      moveJ p935,v100,fine,tool1\WObj:=wobj0;
      moveJ p936,v100,fine,tool1\WObj:=wobj0;
      moveJ p937,v100,fine,tool1\WObj:=wobj0;
      moveJ p938,v100,fine,tool1\WObj:=wobj0;
      moveJ p939,v100,fine,tool1\WObj:=wobj0;
      moveJ p940,v100,fine,tool1\WObj:=wobj0;
      moveJ p941,v100,fine,tool1\WObj:=wobj0;
      moveJ p942,v100,fine,tool1\WObj:=wobj0;
      moveJ p943,v100,fine,tool1\WObj:=wobj0;
      moveJ p944,v100,fine,tool1\WObj:=wobj0;
      moveJ p945,v100,fine,tool1\WObj:=wobj0;
      moveJ p946,v100,fine,tool1\WObj:=wobj0;
      moveJ p947,v100,fine,tool1\WObj:=wobj0;
      moveJ p948,v100,fine,tool1\WObj:=wobj0;
      moveJ p949,v100,fine,tool1\WObj:=wobj0;
      moveJ p950,v100,fine,tool1\WObj:=wobj0;
      moveJ p951,v100,fine,tool1\WObj:=wobj0;
      moveJ p952,v100,fine,tool1\WObj:=wobj0;
      moveJ p953,v100,fine,tool1\WObj:=wobj0;
      moveJ p954,v100,fine,tool1\WObj:=wobj0;
      moveJ p955,v100,fine,tool1\WObj:=wobj0;
      moveJ p956,v100,fine,tool1\WObj:=wobj0;
      moveJ p957,v100,fine,tool1\WObj:=wobj0;
      moveJ p958,v100,fine,tool1\WObj:=wobj0;
      moveJ p959,v100,fine,tool1\WObj:=wobj0;
      moveJ p960,v100,fine,tool1\WObj:=wobj0;
      moveJ p961,v100,fine,tool1\WObj:=wobj0;
      moveJ p962,v100,fine,tool1\WObj:=wobj0;
      moveJ p963,v100,fine,tool1\WObj:=wobj0;
      moveJ p964,v100,fine,tool1\WObj:=wobj0;
      moveJ p965,v100,fine,tool1\WObj:=wobj0;
      moveJ p966,v100,fine,tool1\WObj:=wobj0;
      moveJ p967,v100,fine,tool1\WObj:=wobj0;
      moveJ p968,v100,fine,tool1\WObj:=wobj0;
      moveJ p969,v100,fine,tool1\WObj:=wobj0;
      moveJ p970,v100,fine,tool1\WObj:=wobj0;
      moveJ p971,v100,fine,tool1\WObj:=wobj0;
      moveJ p972,v100,fine,tool1\WObj:=wobj0;
      moveJ p973,v100,fine,tool1\WObj:=wobj0;
      moveJ p974,v100,fine,tool1\WObj:=wobj0;
      moveJ p975,v100,fine,tool1\WObj:=wobj0;
      moveJ p976,v100,fine,tool1\WObj:=wobj0;
      moveJ p977,v100,fine,tool1\WObj:=wobj0;
      moveJ p978,v100,fine,tool1\WObj:=wobj0;
      moveJ p979,v100,fine,tool1\WObj:=wobj0;
      moveJ p980,v100,fine,tool1\WObj:=wobj0;
      moveJ p981,v100,fine,tool1\WObj:=wobj0;
      moveJ p982,v100,fine,tool1\WObj:=wobj0;
      moveJ p983,v100,fine,tool1\WObj:=wobj0;
      moveJ p984,v100,fine,tool1\WObj:=wobj0;
      moveJ p985,v100,fine,tool1\WObj:=wobj0;
      moveJ p986,v100,fine,tool1\WObj:=wobj0;
      moveJ p987,v100,fine,tool1\WObj:=wobj0;
      moveJ p988,v100,fine,tool1\WObj:=wobj0;
      moveJ p989,v100,fine,tool1\WObj:=wobj0;
      moveJ p990,v100,fine,tool1\WObj:=wobj0;
      moveJ p991,v100,fine,tool1\WObj:=wobj0;
      moveJ p992,v100,fine,tool1\WObj:=wobj0;
      moveJ p993,v100,fine,tool1\WObj:=wobj0;
      moveJ p994,v100,fine,tool1\WObj:=wobj0;
      moveJ p995,v100,fine,tool1\WObj:=wobj0;
      moveJ p996,v100,fine,tool1\WObj:=wobj0;
      moveJ p997,v100,fine,tool1\WObj:=wobj0;
      moveJ p998,v100,fine,tool1\WObj:=wobj0;
      moveJ p999,v100,fine,tool1\WObj:=wobj0;
      moveJ p1000,v100,fine,tool1\WObj:=wobj0;
      moveJ p1001,v100,fine,tool1\WObj:=wobj0;
      moveJ p1002,v100,fine,tool1\WObj:=wobj0;
      moveJ p1003,v100,fine,tool1\WObj:=wobj0;
      moveJ p1004,v100,fine,tool1\WObj:=wobj0;
      moveJ p1005,v100,fine,tool1\WObj:=wobj0;
      moveJ p1006,v100,fine,tool1\WObj:=wobj0;
      moveJ p1007,v100,fine,tool1\WObj:=wobj0;
      moveJ p1008,v100,fine,tool1\WObj:=wobj0;
      moveJ p1009,v100,fine,tool1\WObj:=wobj0;
      moveJ p1010,v100,fine,tool1\WObj:=wobj0;
      moveJ p1011,v100,fine,tool1\WObj:=wobj0;
      moveJ p1012,v100,fine,tool1\WObj:=wobj0;
      moveJ p1013,v100,fine,tool1\WObj:=wobj0;
      moveJ p1014,v100,fine,tool1\WObj:=wobj0;
      moveJ p1015,v100,fine,tool1\WObj:=wobj0;
      moveJ p1016,v100,fine,tool1\WObj:=wobj0;
      moveJ p1017,v100,fine,tool1\WObj:=wobj0;
      moveJ p1018,v100,fine,tool1\WObj:=wobj0;
      moveJ p1019,v100,fine,tool1\WObj:=wobj0;
      moveJ p1020,v100,fine,tool1\WObj:=wobj0;
      moveJ p1021,v100,fine,tool1\WObj:=wobj0;
      moveJ p1022,v100,fine,tool1\WObj:=wobj0;
      moveJ p1023,v100,fine,tool1\WObj:=wobj0;
      moveJ p1024,v100,fine,tool1\WObj:=wobj0;
      moveJ p1025,v100,fine,tool1\WObj:=wobj0;
      moveJ p1026,v100,fine,tool1\WObj:=wobj0;
      moveJ p1027,v100,fine,tool1\WObj:=wobj0;
      moveJ p1028,v100,fine,tool1\WObj:=wobj0;
      moveJ p1029,v100,fine,tool1\WObj:=wobj0;
      moveJ p1030,v100,fine,tool1\WObj:=wobj0;
      moveJ p1031,v100,fine,tool1\WObj:=wobj0;
      moveJ p1032,v100,fine,tool1\WObj:=wobj0;
      moveJ p1033,v100,fine,tool1\WObj:=wobj0;
      moveJ p1034,v100,fine,tool1\WObj:=wobj0;
      moveJ p1035,v100,fine,tool1\WObj:=wobj0;
      moveJ p1036,v100,fine,tool1\WObj:=wobj0;
      moveJ p1037,v100,fine,tool1\WObj:=wobj0;
      moveJ p1038,v100,fine,tool1\WObj:=wobj0;
      moveJ p1039,v100,fine,tool1\WObj:=wobj0;
      moveJ p1040,v100,fine,tool1\WObj:=wobj0;
      moveJ p1041,v100,fine,tool1\WObj:=wobj0;
      moveJ p1042,v100,fine,tool1\WObj:=wobj0;
      moveJ p1043,v100,fine,tool1\WObj:=wobj0;
      moveJ p1044,v100,fine,tool1\WObj:=wobj0;
      moveJ p1045,v100,fine,tool1\WObj:=wobj0;
      moveJ p1046,v100,fine,tool1\WObj:=wobj0;
      moveJ p1047,v100,fine,tool1\WObj:=wobj0;
      moveJ p1048,v100,fine,tool1\WObj:=wobj0;
      moveJ p1049,v100,fine,tool1\WObj:=wobj0;
      moveJ p1050,v100,fine,tool1\WObj:=wobj0;
      moveJ p1051,v100,fine,tool1\WObj:=wobj0;
      moveJ p1052,v100,fine,tool1\WObj:=wobj0;
      moveJ p1053,v100,fine,tool1\WObj:=wobj0;
      moveJ p1054,v100,fine,tool1\WObj:=wobj0;
      moveJ p1055,v100,fine,tool1\WObj:=wobj0;
      moveJ p1056,v100,fine,tool1\WObj:=wobj0;
      moveJ p1057,v100,fine,tool1\WObj:=wobj0;
      moveJ p1058,v100,fine,tool1\WObj:=wobj0;
      moveJ p1059,v100,fine,tool1\WObj:=wobj0;
      moveJ p1060,v100,fine,tool1\WObj:=wobj0;
      moveJ p1061,v100,fine,tool1\WObj:=wobj0;
      moveJ p1062,v100,fine,tool1\WObj:=wobj0;
      moveJ p1063,v100,fine,tool1\WObj:=wobj0;
      moveJ p1064,v100,fine,tool1\WObj:=wobj0;
      moveJ p1065,v100,fine,tool1\WObj:=wobj0;
      moveJ p1066,v100,fine,tool1\WObj:=wobj0;
      moveJ p1067,v100,fine,tool1\WObj:=wobj0;
      moveJ p1068,v100,fine,tool1\WObj:=wobj0;
      moveJ p1069,v100,fine,tool1\WObj:=wobj0;
      moveJ p1070,v100,fine,tool1\WObj:=wobj0;
      moveJ p1071,v100,fine,tool1\WObj:=wobj0;
      moveJ p1072,v100,fine,tool1\WObj:=wobj0;
      moveJ p1073,v100,fine,tool1\WObj:=wobj0;
      moveJ p1074,v100,fine,tool1\WObj:=wobj0;
      moveJ p1075,v100,fine,tool1\WObj:=wobj0;
      moveJ p1076,v100,fine,tool1\WObj:=wobj0;
      moveJ p1077,v100,fine,tool1\WObj:=wobj0;
      moveJ p1078,v100,fine,tool1\WObj:=wobj0;
      moveJ p1079,v100,fine,tool1\WObj:=wobj0;
      moveJ p1080,v100,fine,tool1\WObj:=wobj0;
      moveJ p1081,v100,fine,tool1\WObj:=wobj0;
      moveJ p1082,v100,fine,tool1\WObj:=wobj0;
      moveJ p1083,v100,fine,tool1\WObj:=wobj0;
      moveJ p1084,v100,fine,tool1\WObj:=wobj0;
      moveJ p1085,v100,fine,tool1\WObj:=wobj0;
      moveJ p1086,v100,fine,tool1\WObj:=wobj0;
      moveJ p1087,v100,fine,tool1\WObj:=wobj0;
      moveJ p1088,v100,fine,tool1\WObj:=wobj0;
      moveJ p1089,v100,fine,tool1\WObj:=wobj0;
      moveJ p1090,v100,fine,tool1\WObj:=wobj0;
      moveJ p1091,v100,fine,tool1\WObj:=wobj0;
      moveJ p1092,v100,fine,tool1\WObj:=wobj0;
      moveJ p1093,v100,fine,tool1\WObj:=wobj0;
      moveJ p1094,v100,fine,tool1\WObj:=wobj0;
      moveJ p1095,v100,fine,tool1\WObj:=wobj0;
      moveJ p1096,v100,fine,tool1\WObj:=wobj0;
      moveJ p1097,v100,fine,tool1\WObj:=wobj0;
      moveJ p1098,v100,fine,tool1\WObj:=wobj0;
      moveJ p1099,v100,fine,tool1\WObj:=wobj0;
      moveJ p1100,v100,fine,tool1\WObj:=wobj0;
      moveJ p1101,v100,fine,tool1\WObj:=wobj0;
      moveJ p1102,v100,fine,tool1\WObj:=wobj0;
      moveJ p1103,v100,fine,tool1\WObj:=wobj0;
      moveJ p1104,v100,fine,tool1\WObj:=wobj0;
      moveJ p1105,v100,fine,tool1\WObj:=wobj0;
      moveJ p1106,v100,fine,tool1\WObj:=wobj0;
      moveJ p1107,v100,fine,tool1\WObj:=wobj0;
      moveJ p1108,v100,fine,tool1\WObj:=wobj0;
      moveJ p1109,v100,fine,tool1\WObj:=wobj0;
      moveJ p1110,v100,fine,tool1\WObj:=wobj0;
      moveJ p1111,v100,fine,tool1\WObj:=wobj0;
      moveJ p1112,v100,fine,tool1\WObj:=wobj0;
      moveJ p1113,v100,fine,tool1\WObj:=wobj0;
      moveJ p1114,v100,fine,tool1\WObj:=wobj0;
      moveJ p1115,v100,fine,tool1\WObj:=wobj0;
      moveJ p1116,v100,fine,tool1\WObj:=wobj0;
      moveJ p1117,v100,fine,tool1\WObj:=wobj0;
      moveJ p1118,v100,fine,tool1\WObj:=wobj0;
      moveJ p1119,v100,fine,tool1\WObj:=wobj0;
      moveJ p1120,v100,fine,tool1\WObj:=wobj0;
      moveJ p1121,v100,fine,tool1\WObj:=wobj0;
      moveJ p1122,v100,fine,tool1\WObj:=wobj0;
      moveJ p1123,v100,fine,tool1\WObj:=wobj0;
      moveJ p1124,v100,fine,tool1\WObj:=wobj0;
      moveJ p1125,v100,fine,tool1\WObj:=wobj0;
      moveJ p1126,v100,fine,tool1\WObj:=wobj0;
      moveJ p1127,v100,fine,tool1\WObj:=wobj0;
      moveJ p1128,v100,fine,tool1\WObj:=wobj0;
      moveJ p1129,v100,fine,tool1\WObj:=wobj0;
      moveJ p1130,v100,fine,tool1\WObj:=wobj0;
      moveJ p1131,v100,fine,tool1\WObj:=wobj0;
      moveJ p1132,v100,fine,tool1\WObj:=wobj0;
      moveJ p1133,v100,fine,tool1\WObj:=wobj0;
      moveJ p1134,v100,fine,tool1\WObj:=wobj0;
      moveJ p1135,v100,fine,tool1\WObj:=wobj0;
      moveJ p1136,v100,fine,tool1\WObj:=wobj0;
      moveJ p1137,v100,fine,tool1\WObj:=wobj0;
      moveJ p1138,v100,fine,tool1\WObj:=wobj0;
      moveJ p1139,v100,fine,tool1\WObj:=wobj0;
      moveJ p1140,v100,fine,tool1\WObj:=wobj0;
      moveJ p1141,v100,fine,tool1\WObj:=wobj0;
      moveJ p1142,v100,fine,tool1\WObj:=wobj0;
      moveJ p1143,v100,fine,tool1\WObj:=wobj0;
      moveJ p1144,v100,fine,tool1\WObj:=wobj0;
      moveJ p1145,v100,fine,tool1\WObj:=wobj0;
      moveJ p1146,v100,fine,tool1\WObj:=wobj0;
      moveJ p1147,v100,fine,tool1\WObj:=wobj0;
      moveJ p1148,v100,fine,tool1\WObj:=wobj0;
      moveJ p1149,v100,fine,tool1\WObj:=wobj0;
      moveJ p1150,v100,fine,tool1\WObj:=wobj0;
      moveJ p1151,v100,fine,tool1\WObj:=wobj0;
      moveJ p1152,v100,fine,tool1\WObj:=wobj0;
      moveJ p1153,v100,fine,tool1\WObj:=wobj0;
      moveJ p1154,v100,fine,tool1\WObj:=wobj0;
      moveJ p1155,v100,fine,tool1\WObj:=wobj0;
      moveJ p1156,v100,fine,tool1\WObj:=wobj0;
      moveJ p1157,v100,fine,tool1\WObj:=wobj0;
      moveJ p1158,v100,fine,tool1\WObj:=wobj0;
      moveJ p1159,v100,fine,tool1\WObj:=wobj0;
      moveJ p1160,v100,fine,tool1\WObj:=wobj0;
      moveJ p1161,v100,fine,tool1\WObj:=wobj0;
      moveJ p1162,v100,fine,tool1\WObj:=wobj0;
      moveJ p1163,v100,fine,tool1\WObj:=wobj0;
      moveJ p1164,v100,fine,tool1\WObj:=wobj0;
      moveJ p1165,v100,fine,tool1\WObj:=wobj0;
      moveJ p1166,v100,fine,tool1\WObj:=wobj0;
      moveJ p1167,v100,fine,tool1\WObj:=wobj0;
      moveJ p1168,v100,fine,tool1\WObj:=wobj0;
      moveJ p1169,v100,fine,tool1\WObj:=wobj0;
      moveJ p1170,v100,fine,tool1\WObj:=wobj0;
      moveJ p1171,v100,fine,tool1\WObj:=wobj0;
      moveJ p1172,v100,fine,tool1\WObj:=wobj0;
      moveJ p1173,v100,fine,tool1\WObj:=wobj0;
      moveJ p1174,v100,fine,tool1\WObj:=wobj0;
      moveJ p1175,v100,fine,tool1\WObj:=wobj0;
      moveJ p1176,v100,fine,tool1\WObj:=wobj0;
      moveJ p1177,v100,fine,tool1\WObj:=wobj0;
      moveJ p1178,v100,fine,tool1\WObj:=wobj0;
      moveJ p1179,v100,fine,tool1\WObj:=wobj0;
      moveJ p1180,v100,fine,tool1\WObj:=wobj0;
      moveJ p1181,v100,fine,tool1\WObj:=wobj0;
      moveJ p1182,v100,fine,tool1\WObj:=wobj0;
      moveJ p1183,v100,fine,tool1\WObj:=wobj0;
      moveJ p1184,v100,fine,tool1\WObj:=wobj0;
      moveJ p1185,v100,fine,tool1\WObj:=wobj0;
      moveJ p1186,v100,fine,tool1\WObj:=wobj0;
      moveJ p1187,v100,fine,tool1\WObj:=wobj0;
      moveJ p1188,v100,fine,tool1\WObj:=wobj0;
      moveJ p1189,v100,fine,tool1\WObj:=wobj0;
      moveJ p1190,v100,fine,tool1\WObj:=wobj0;
      moveJ p1191,v100,fine,tool1\WObj:=wobj0;
      moveJ p1192,v100,fine,tool1\WObj:=wobj0;
      moveJ p1193,v100,fine,tool1\WObj:=wobj0;
      moveJ p1194,v100,fine,tool1\WObj:=wobj0;
      moveJ p1195,v100,fine,tool1\WObj:=wobj0;
      moveJ p1196,v100,fine,tool1\WObj:=wobj0;
      moveJ p1197,v100,fine,tool1\WObj:=wobj0;
      moveJ p1198,v100,fine,tool1\WObj:=wobj0;
      moveJ p1199,v100,fine,tool1\WObj:=wobj0;
      moveJ p1200,v100,fine,tool1\WObj:=wobj0;
      moveJ p1201,v100,fine,tool1\WObj:=wobj0;
      moveJ p1202,v100,fine,tool1\WObj:=wobj0;
      moveJ p1203,v100,fine,tool1\WObj:=wobj0;
      moveJ p1204,v100,fine,tool1\WObj:=wobj0;
      moveJ p1205,v100,fine,tool1\WObj:=wobj0;
      moveJ p1206,v100,fine,tool1\WObj:=wobj0;
      moveJ p1207,v100,fine,tool1\WObj:=wobj0;
      moveJ p1208,v100,fine,tool1\WObj:=wobj0;
      moveJ p1209,v100,fine,tool1\WObj:=wobj0;
      moveJ p1210,v100,fine,tool1\WObj:=wobj0;
      moveJ p1211,v100,fine,tool1\WObj:=wobj0;
      moveJ p1212,v100,fine,tool1\WObj:=wobj0;
      moveJ p1213,v100,fine,tool1\WObj:=wobj0;
      moveJ p1214,v100,fine,tool1\WObj:=wobj0;
      moveJ p1215,v100,fine,tool1\WObj:=wobj0;
      moveJ p1216,v100,fine,tool1\WObj:=wobj0;
      moveJ p1217,v100,fine,tool1\WObj:=wobj0;
      moveJ p1218,v100,fine,tool1\WObj:=wobj0;
      moveJ p1219,v100,fine,tool1\WObj:=wobj0;
      moveJ p1220,v100,fine,tool1\WObj:=wobj0;
      moveJ p1221,v100,fine,tool1\WObj:=wobj0;
      moveJ p1222,v100,fine,tool1\WObj:=wobj0;
      moveJ p1223,v100,fine,tool1\WObj:=wobj0;
      moveJ p1224,v100,fine,tool1\WObj:=wobj0;
      moveJ p1225,v100,fine,tool1\WObj:=wobj0;
      moveJ p1226,v100,fine,tool1\WObj:=wobj0;
      moveJ p1227,v100,fine,tool1\WObj:=wobj0;
      moveJ p1228,v100,fine,tool1\WObj:=wobj0;
      moveJ p1229,v100,fine,tool1\WObj:=wobj0;
      moveJ p1230,v100,fine,tool1\WObj:=wobj0;
      moveJ p1231,v100,fine,tool1\WObj:=wobj0;
      moveJ p1232,v100,fine,tool1\WObj:=wobj0;
      moveJ p1233,v100,fine,tool1\WObj:=wobj0;
      moveJ p1234,v100,fine,tool1\WObj:=wobj0;
      moveJ p1235,v100,fine,tool1\WObj:=wobj0;
      moveJ p1236,v100,fine,tool1\WObj:=wobj0;
      moveJ p1237,v100,fine,tool1\WObj:=wobj0;
      moveJ p1238,v100,fine,tool1\WObj:=wobj0;
      moveJ p1239,v100,fine,tool1\WObj:=wobj0;
      moveJ p1240,v100,fine,tool1\WObj:=wobj0;
      moveJ p1241,v100,fine,tool1\WObj:=wobj0;
      moveJ p1242,v100,fine,tool1\WObj:=wobj0;
      moveJ p1243,v100,fine,tool1\WObj:=wobj0;
      moveJ p1244,v100,fine,tool1\WObj:=wobj0;
      moveJ p1245,v100,fine,tool1\WObj:=wobj0;
      moveJ p1246,v100,fine,tool1\WObj:=wobj0;
      moveJ p1247,v100,fine,tool1\WObj:=wobj0;
      moveJ p1248,v100,fine,tool1\WObj:=wobj0;
      moveJ p1249,v100,fine,tool1\WObj:=wobj0;
      moveJ p1250,v100,fine,tool1\WObj:=wobj0;
      moveJ p1251,v100,fine,tool1\WObj:=wobj0;
      moveJ p1252,v100,fine,tool1\WObj:=wobj0;
      moveJ p1253,v100,fine,tool1\WObj:=wobj0;
      moveJ p1254,v100,fine,tool1\WObj:=wobj0;
      moveJ p1255,v100,fine,tool1\WObj:=wobj0;
      moveJ p1256,v100,fine,tool1\WObj:=wobj0;
      moveJ p1257,v100,fine,tool1\WObj:=wobj0;
      moveJ p1258,v100,fine,tool1\WObj:=wobj0;
      moveJ p1259,v100,fine,tool1\WObj:=wobj0;
      moveJ p1260,v100,fine,tool1\WObj:=wobj0;
      moveJ p1261,v100,fine,tool1\WObj:=wobj0;
      moveJ p1262,v100,fine,tool1\WObj:=wobj0;
      moveJ p1263,v100,fine,tool1\WObj:=wobj0;
      moveJ p1264,v100,fine,tool1\WObj:=wobj0;
      moveJ p1265,v100,fine,tool1\WObj:=wobj0;
      moveJ p1266,v100,fine,tool1\WObj:=wobj0;
      moveJ p1267,v100,fine,tool1\WObj:=wobj0;
      moveJ p1268,v100,fine,tool1\WObj:=wobj0;
      moveJ p1269,v100,fine,tool1\WObj:=wobj0;
      moveJ p1270,v100,fine,tool1\WObj:=wobj0;
      moveJ p1271,v100,fine,tool1\WObj:=wobj0;
      moveJ p1272,v100,fine,tool1\WObj:=wobj0;
      moveJ p1273,v100,fine,tool1\WObj:=wobj0;
      moveJ p1274,v100,fine,tool1\WObj:=wobj0;
      moveJ p1275,v100,fine,tool1\WObj:=wobj0;
      moveJ p1276,v100,fine,tool1\WObj:=wobj0;
      moveJ p1277,v100,fine,tool1\WObj:=wobj0;
      moveJ p1278,v100,fine,tool1\WObj:=wobj0;
      moveJ p1279,v100,fine,tool1\WObj:=wobj0;
      moveJ p1280,v100,fine,tool1\WObj:=wobj0;
      moveJ p1281,v100,fine,tool1\WObj:=wobj0;
      moveJ p1282,v100,fine,tool1\WObj:=wobj0;
      moveJ p1283,v100,fine,tool1\WObj:=wobj0;
      moveJ p1284,v100,fine,tool1\WObj:=wobj0;
      moveJ p1285,v100,fine,tool1\WObj:=wobj0;
      moveJ p1286,v100,fine,tool1\WObj:=wobj0;
      moveJ p1287,v100,fine,tool1\WObj:=wobj0;
      moveJ p1288,v100,fine,tool1\WObj:=wobj0;
      moveJ p1289,v100,fine,tool1\WObj:=wobj0;
      moveJ p1290,v100,fine,tool1\WObj:=wobj0;
      moveJ p1291,v100,fine,tool1\WObj:=wobj0;
      moveJ p1292,v100,fine,tool1\WObj:=wobj0;
      moveJ p1293,v100,fine,tool1\WObj:=wobj0;
      moveJ p1294,v100,fine,tool1\WObj:=wobj0;
      moveJ p1295,v100,fine,tool1\WObj:=wobj0;
      moveJ p1296,v100,fine,tool1\WObj:=wobj0;
      moveJ p1297,v100,fine,tool1\WObj:=wobj0;
      moveJ p1298,v100,fine,tool1\WObj:=wobj0;
      moveJ p1299,v100,fine,tool1\WObj:=wobj0;
      moveJ p1300,v100,fine,tool1\WObj:=wobj0;
   ENDPROC
ENDMODULE
